// Mitsubishi GX Works2 project: word_bitcontrol   PLC: Q02/Q02H

PROGRAM MAIN
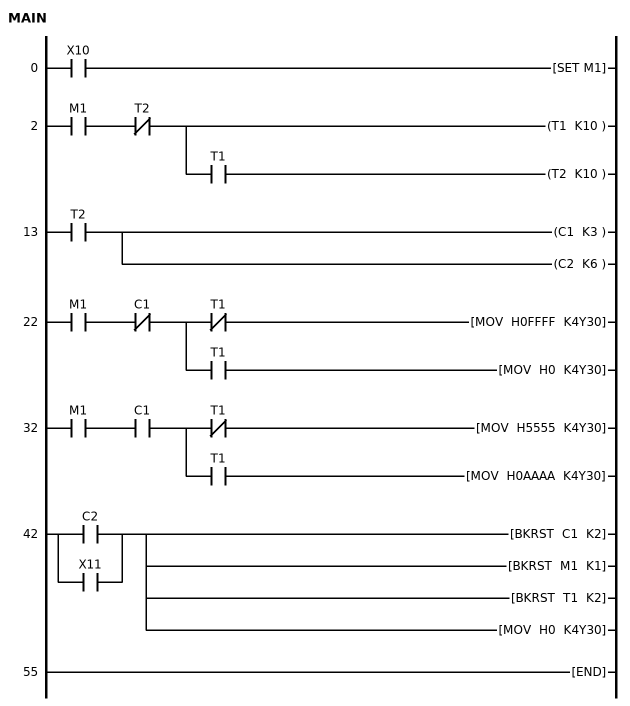
0     LD      X10
      SET     M1
2     LD      M1
      ANI     T2
      OUT     T1 K10
      AND     T1
      OUT     T2 K10
13    LD      T2
      OUT     C1 K3
      OUT     C2 K6
22    LD      M1
      ANI     C1
      MPS
      ANI     T1
      MOV     H0FFFF K4Y30
      MPP
      AND     T1
      MOV     H0 K4Y30
32    LD      M1
      AND     C1
      MPS
      ANI     T1
      MOV     H5555 K4Y30
      MPP
      AND     T1
      MOV     H0AAAA K4Y30
42    LD      C2
      OR      X11
      BKRST   C1 K2
      BKRST   M1 K1
      BKRST   T1 K2
      MOV     H0 K4Y30
55    END
END_PROGRAM

PROGRAM operand
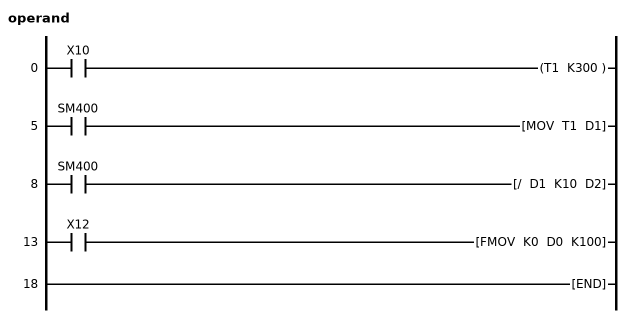
0     LD      X10
      OUT     T1 K300
5     LD      SM400
      MOV     T1 D1
8     LD      SM400
      /       D1 K10 D2
13    LD      X12
      FMOV    K0 D0 K100
18    END
END_PROGRAM

PROGRAM compare
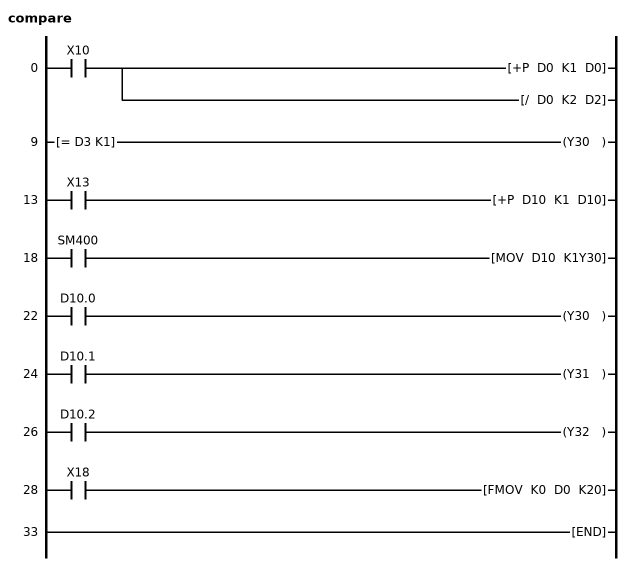
0     LD      X10
      +P      D0 K1 D0
      /       D0 K2 D2
9     LD=     D3 K1
      OUT     Y30
13    LD      X13
      +P      D10 K1 D10
18    LD      SM400
      MOV     D10 K1Y30
22    LD      D10.0
      OUT     Y30
24    LD      D10.1
      OUT     Y31
26    LD      D10.2
      OUT     Y32
28    LD      X18
      FMOV    K0 D0 K20
33    END
END_PROGRAM
